FUNCTION_BLOCK FB_Observable_USINT EXTENDS FB_AbstractObservable
VAR
    _nVal:              USINT;
    _nOldVal:           USINT;
END_VAR

METHOD FB_init : BOOL
VAR_INPUT
    bInitRetains:       BOOL; // if TRUE, the retain variables are initialized (warm start / cold start)
    bInCopyCode:        BOOL;  // if TRUE, the instance afterwards gets moved into the copy code (online change)
END_VAR
THIS^._nTypeClass := __SYSTEM.TYPE_CLASS.TYPE_USINT;
END_METHOD

PROPERTY nDataSize : UDINT
GET
nDataSize := SIZEOF(USINT);
END_GET
END_PROPERTY

PROPERTY nValue8 : USINT
GET
nValue8 := THIS^._nVal;
END_GET
SET
THIS^._nOldVal := THIS^._nVal;
THIS^._nVal := nValue8;

THIS^.NotifyWithConditions();
END_SET
END_PROPERTY

PROPERTY PROTECTED pData : POINTER TO BYTE
GET
pData := ADR(THIS^._nVal);
END_GET
END_PROPERTY

METHOD  ValueChanged : BOOL
VAR_INPUT
END_VAR
ValueChanged := THIS^._nOldVal <> THIS^._nVal;
END_METHOD

END_FUNCTION_BLOCK

(* stored: Version 1.1.0.1, ProductVersion 3.1.4024.12
   POU FB_Observable_USINT: Id {df32fa4f-80a2-0fa3-3ffb-2809d40a7d2a}, SpecialFunc None
   Method FB_init: Id {404da6a5-566c-0b67-11b8-31fecbba6568}
   Property nDataSize: Id {059688f0-64f3-0350-3ac4-3e40872834c4}
   Get Get: Id {d6e9f9e1-2955-03c1-1cca-aa8a89faffd9}
   Property nValue8: Id {943b19d9-d338-0d9d-162c-969292bc534b}
   Get Get: Id {017c5fac-b6a8-0cab-2206-a9ce52cb44aa}
   Set Set: Id {c62a7ebc-f1de-08bf-0fbc-5e9f63399214}
   Property pData: Id {8163fc7a-17da-095d-2b49-3602f8b6e9a3}
   Get Get: Id {be9f7aa0-2bb9-0e91-3052-825e4cb778a7}
   Method ValueChanged: Id {31bddad3-f54e-0545-1dbd-644c94ec8e67} *)
